{attribute 'qualified_only'}
{attribute 'strict'}
TYPE E_EncoderType :
(
	Incremental := 0 ,
	Absolute := 1
);
END_TYPE

(* stored: Version 1.1.0.1, ProductVersion 3.1.4024.3
   DUT E_EncoderType: Id {83ddf9c4-2f65-4a7b-8d10-700800b033f1} *)
